// TIA Portal V21 export
FUNCTION_BLOCK "AlarmsContainer"   // FB200, LAD
{ S7_Optimized_Access := 'TRUE' }
// stored: AutoNumber false, MemoryReserve 100, SetENOAutomatically false
   VAR
      WeeklyReset { ExternalAccessible := 'False'; ExternalVisible := 'False'; ExternalWritable := 'False'} : Bool;
      MaintenanceReset : Bool;
      Edge { ExternalAccessible := 'False'; ExternalVisible := 'False'; ExternalWritable := 'False'} : Array[0..10] of Bool;
   END_VAR
   VAR_TEMP
      tempBool : Bool;
      i : USInt;
      j : USInt;
      n : DInt;
      Addr : DInt;
   END_VAR
   VAR_TEMP   // added for the SCL form of the ladder/FBD networks
      _w1 : Bool;
   END_VAR
BEGIN

REGION Network 1: ======================================= General
END_REGION

REGION Network 2: Emergency stop
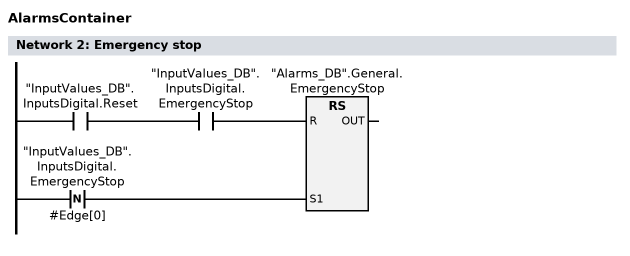
   RUNG wire#powerrail
      Contact( "InputValues_DB".InputsDigital.Reset )
      Contact( "InputValues_DB".InputsDigital.EmergencyStop )
      S_RS(operand := "Alarms_DB".General.EmergencyStop, s1 := wire#w1)
   END_RUNG
   RUNG wire#powerrail
      N_Contact(operand := "InputValues_DB".InputsDigital.EmergencyStop, bit := #Edge[0])
   END_RUNG wire#w1
   // the same network as SCL:
   #_w1 := NOT "InputValues_DB".InputsDigital.EmergencyStop AND #Edge[0];   // falling edge of "InputValues_DB".InputsDigital.EmergencyStop
   #Edge[0] := "InputValues_DB".InputsDigital.EmergencyStop;
   IF "InputValues_DB".InputsDigital.Reset AND "InputValues_DB".InputsDigital.EmergencyStop THEN
       "Alarms_DB".General.EmergencyStop := FALSE;   // RS flip-flop
   END_IF;
   IF #_w1 THEN "Alarms_DB".General.EmergencyStop := TRUE; END_IF;
END_REGION

REGION Network 3 (SCL): ======================================= PLC
   // TODO
   FOR #i := 2 TO 5 DO
       IF #i = 2 THEN
           #Addr := 200;
           #n := 0;
       ELSIF #i = 4 THEN
           #Addr := 204;
           #n := 0;
       END_IF;
       FOR #j := 0 TO 7 DO
           #tempBool := PEEK_BOOL(area := 16#81, dbNumber := 0, byteOffset := #Addr + #n, bitOffset := #j);
           IF NOT #tempBool THEN
               POKE_BOOL(area := 16#84,
                         dbNumber := 201,
                         byteOffset := #i,
                         bitOffset := #j,
                         value := TRUE);
           ELSIF "InputValues_DB".InputsDigital.Reset THEN
               POKE_BOOL(area := 16#84,
                         dbNumber := 201,
                         byteOffset := #i,
                         bitOffset := #j,
                         value := FALSE);
           END_IF;
       END_FOR;
       #n += 1;
   END_FOR;
END_REGION
END_FUNCTION_BLOCK
